// TwinCAT 3 PLC project PLC_Test
// ProgramVersion: 3.1.4024.0
// libraries:
//   Tc2_Standard, * (Beckhoff Automation GmbH)
//   Tc2_System, * (Beckhoff Automation GmbH)
//   Tc3_Module, * (Beckhoff Automation GmbH)
// project tree:
//   / GlobalTextList.TcGTLO, PlcTask.TcTTO, Visualization Manager.TcVMO (not stored)
//   POUs/ MAIN.TcPOU, Q5.TcPOU, Q1.TcPOU, Q2.TcPOU, Q3.TcPOU, Q4.TcPOU, Q6.TcPOU, Q7.TcPOU
//   VISUs/ Q7_V.TcVIS
// real-time tasks:
//   TASK PlcTask: cycle T#10ms, priority 20, ADS port 350

CONFIGURATION PLC_Test
    RESOURCE PLC ON TwinCAT3
        TASK PlcTask(INTERVAL := T#10ms, PRIORITY := 20);
        PROGRAM MAIN WITH PlcTask : MAIN;
    END_RESOURCE
END_CONFIGURATION

// ---- POUs/MAIN.TcPOU
PROGRAM MAIN
VAR
END_VAR

// Code also available on my GitHub (will make it public after the test closes)
// https://github.com/JPChurchouse/282762_PLCs/tree/main/Test

//Q3(); // Uncomment to run Question Three
//Q4(); // Uncomment to run Question Four
Q7(); // Uncomment to run Question Seven

END_PROGRAM

// ---- POUs/Q7.TcPOU
PROGRAM Q7
VAR
	button_up 	: BOOL 	:= FALSE;
	moving		: BOOL 	:= FALSE;
	
END_VAR

// When the up button is pressed, the moving status indicator will toggle

// To run this program, paste the following into MAIN, then interact with the Visualisation Q7_V
// Q7();
VAR // added by the converter: edge detectors and wires of the graphical bodies
    _w1 : BOOL;
END_VAR

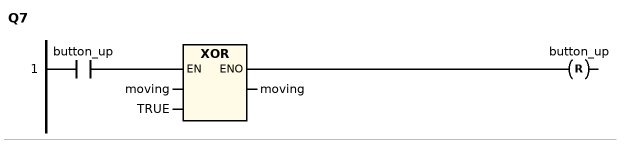
// NETWORK 1
_w1 := button_up;
IF _w1 THEN moving := moving XOR TRUE; END_IF
button_up R= _w1;

END_PROGRAM

// ---- POUs/Q5.TcPOU
PROGRAM Q5
VAR
	i : INT := 0;
 	output : BOOL := FALSE;
END_VAR

(*
init:
	i is an INT init to 0
	output is a BOOL init to false

1:
	0 is assigned to i
	
	i == 0
	
2:
	if i > 0, not goto label default
	
	i is not > 0, therefore goto -> default:
	
3:
	TRUE is assigned to output
	
	not executed as it was jumped by the goto label

4:
	label default, no functionality
	
	no functionality, return
	
end:
	output has value FALSE at the end of execution

*)

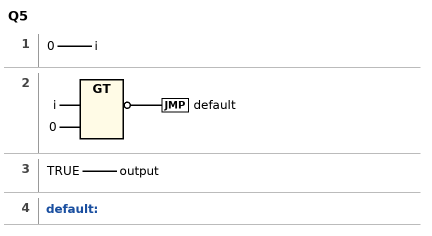
// NETWORK 1
i := 0;

// NETWORK 2
IF NOT (i > 0) THEN JMP default; END_IF

// NETWORK 3
output := TRUE;

// NETWORK 4
default: ;

END_PROGRAM

// ---- POUs/Q1.TcPOU
PROGRAM Q1
VAR
END_VAR

(*
LLD, Ladder Logic Diagram
Each function or state can be put into it's own Network.
These Networks are usually activated while a BOOL is true, and usually sets or resets another BOOL at the end.

Advantages include:
	Easy and quick to learn / implement
	Easy to read
	Graphical logic display rather than text
	
Disadvantages include:
	More intricate operations are a bit tricky to implement
	All Networks are executed concurrently so states must be represented by BOOLs
	

*)

// NETWORK 1

END_PROGRAM

// ---- POUs/Q2.TcPOU
PROGRAM Q2
VAR
END_VAR

(*
SFC, Sequential Function Chart
Operations are represented with states that have transition conditions (hence Sequntial)
Operations are run whilst the containing state is active

Advantages include:
	Easy to get basic states implemented
	Transition conditions are very clear
	May have operations on the entry or exit of a state
	
Disadvantages include:
	More intricate operations are a bit tricky to implement
	Concurrent operations are more difficult or repetitive to implement

*)

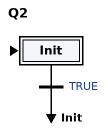
INITIAL_STEP Init:
END_STEP
TRANSITION FROM Init TO Init
    := TRUE;
END_TRANSITION

END_PROGRAM

// ---- POUs/Q3.TcPOU
PROGRAM Q3
VAR
	S1 : BOOL := FALSE; // First Switch
	S2 : BOOL := FALSE; // Second Switch
	M1 : BOOL := FALSE; // Motor
END_VAR

// To run:
// Paste the following into the MAIN file
// Q3();

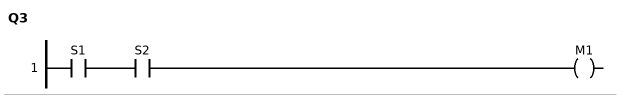
// NETWORK 1
M1 := S1 AND S2;

END_PROGRAM

// ---- POUs/Q4.TcPOU
PROGRAM Q4
VAR
	time_on : TIME := T#1S; 	//On for One second
	time_off : TIME := T#5S;	// Off for five seconds
	L1 : BOOL := FALSE;			// Represents the output
	TON_0: TON;
	TON_1: TON;
END_VAR

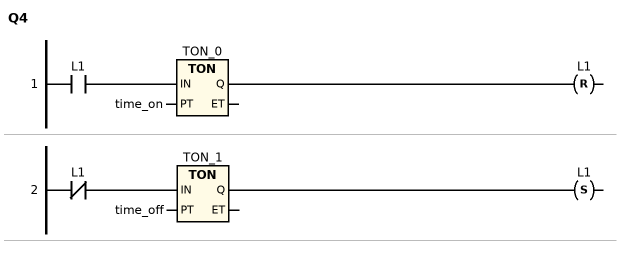
// NETWORK 1
TON_0(IN := L1, PT := time_on); // TON
L1 R= TON_0.Q;

// NETWORK 2
TON_1(IN := NOT L1, PT := time_off); // TON
L1 S= TON_1.Q;

END_PROGRAM

// ---- POUs/Q6.TcPOU
PROGRAM Q6
VAR
	// Parts present?
	partA : BOOL := FALSE;
	partB : BOOL := FALSE;	
	
	// Button pressed?
	button : BOOL := FALSE;
	
	// Running operation
	TON_0: TON;
	time_ext : TIME := T#1S;
	extend : BOOL := FALSE;
	
	// Transition flags
	start: BOOL := FALSE;
	complete : BOOL := FALSE;
	
END_VAR

// BSOD recovery @ 1447hrs

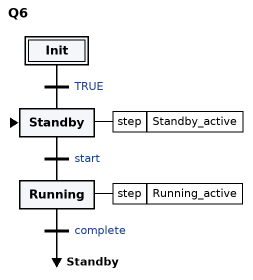
INITIAL_STEP Init:
END_STEP
TRANSITION FROM Init TO Standby
    := TRUE;
END_TRANSITION
STEP Standby:
    Standby_active(N);  // step action
END_STEP
TRANSITION FROM Standby TO Running
    := start;
END_TRANSITION
STEP Running:
    Running_active(N);  // step action
END_STEP
TRANSITION FROM Running TO Standby
    := complete;
END_TRANSITION

ACTION Running_active:
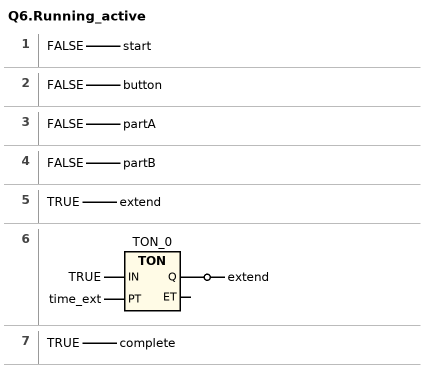
// NETWORK 1
start := FALSE;

// NETWORK 2
button := FALSE;

// NETWORK 3
partA := FALSE;

// NETWORK 4
partB := FALSE;

// NETWORK 5
extend := TRUE;

// NETWORK 6
TON_0(IN := TRUE, PT := time_ext); // TON
extend := NOT TON_0.Q;

// NETWORK 7
complete := TRUE;
END_ACTION

ACTION Standby_active:
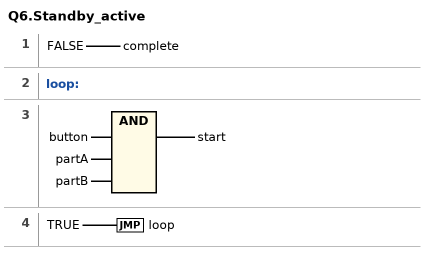
// NETWORK 1
complete := FALSE;

// NETWORK 2
loop: ;

// NETWORK 3
start := button AND partA AND partB;

// NETWORK 4
JMP loop;
END_ACTION

END_PROGRAM

// ---- GlobalTextList.TcGTLO
TEXTLIST GlobalTextList
  868 = '/\\'
  224 = 'Acsend'
  921 = 'Ascend'
  737 = 'At the Bottom'
  156 = 'At the top'
  238 = 'At the Top'
  536 = 'Currently Moving'
  246 = 'Decend'
  87 = 'Descend'
  840 = 'Direction'
  283 = 'Eleveator Status'
  733 = '\\/'
END_TEXTLIST

// ---- VISUs/Q7_V.TcVIS
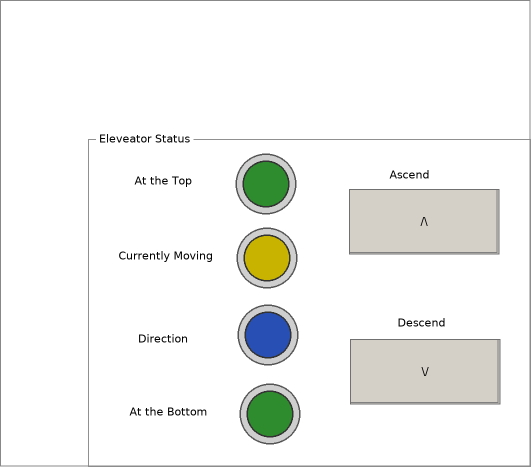
VISUALIZATION Q7_V  // 531x467
    GroupBox (88,131 443x336), "Eleveator Status"
        Lamp1 (143,18 70x70), style: Lamp-Lamp1-Green
        Lamp1 (144,92 70x70), variable: Q7.moving, style: Lamp-Lamp1-Yellow
        Lamp1 (145,169 70x70), variable: true, style: Lamp-Lamp1-Blue
        Lamp1 (147,248 70x70), style: Lamp-Lamp1-Green
        Button (261,58 150x65), "/\"
            OnMouseClick: execute { Q7.button_up := TRUE }
        Button (262,208 150x65), "\/"
        Label (286,177 95x30), "Descend"
        Label (277,29 89x30), "Ascend"
        Label (25,193 100x30), "Direction"
        Label (29,266 103x30), "At the Bottom"
        Label (27,35 97x30), "At the Top"
        Label (25,110 106x30), "Currently Moving"
END_VISUALIZATION
